Fanuc KAREL source: app_abort.kl

PROGRAM appabort

%COMMENT = 'appabort v1'
%NOLOCKGROUP
%NOBUSYLAMP

VAR
	rf_ :FILE
	STATUS: INTEGER

BEGIN

	OPEN FILE rf_ ('RW', 'RD:RESPONSE.HTM')
	STATUS = IO_STATUS(rf_)
	IF (STATUS <> 0) THEN
		WRITE rf_ ( '{"result":"failed", "program":"appabort", "reason":',STATUS,'}')
	ELSE
		WRITE rf_ ( '{"result":"success", "program":"appabort", "reason":',STATUS,'}')
	ENDIF
	CLOSE FILE rf_
	ABORT_TASK('*ALL*', TRUE, TRUE, STATUS)
END appabort
